FUNCTION_BLOCK Test_RaiseNotification_CallsMethod EXTENDS tcl_SimpleUnitTestLibrary.T_UnitTestBase
VAR
    Source  : T_ClassThatRaisesNotifications;
    Handler : T_ClassThatHandlesNotifications;
END_VAR

Handler.FB_init(
    bInitRetains := FALSE,  
    bInCopyCode  := FALSE);

Source.OnPressedNotification.ClearNotificationHandlers();
Source.OnPressedNotification.AddNotificationHandler(Handler);

Source.RaiseOnPbPressedNotification();

Assertion.AssertEquals_UDINT(
    Expected     := 1,
    Actual       := Handler.NotificationCallCount,
    VariableName := 'Dispatcher.NotificationCount');

TestFinished();

END_FUNCTION_BLOCK

(* stored: Version 1.1.0.1, ProductVersion 3.1.4024.4
   POU Test_RaiseNotification_CallsMethod: Id {cc5ef7a4-9804-419b-b45f-a2befe39c1e5}, SpecialFunc None *)
